FUNCTION_BLOCK NodePack_PlcBasic IMPLEMENTS I_NodePack
VAR
	nodePack_PlcBasicDisplay : NodePack_PlcBasicDisplay;
	nodePack_PlcBasicLiterals : NodePack_PlcBasicLiterals;
END_VAR

METHOD PUBLIC RegisterWithNodeFactory
VAR_INPUT
	NodeFactory : I_NodeFactory;
END_VAR
nodePack_PlcBasicDisplay.RegisterWithNodeFactory(NodeFactory);
nodePack_PlcBasicLiterals.RegisterWithNodeFactory(NodeFactory);
END_METHOD

END_FUNCTION_BLOCK

(* stored: Version 1.1.0.1, ProductVersion 3.1.4024.12
   POU NodePack_PlcBasic: Id {b1a7208c-fa6a-0ca2-104f-e5f6ddafa07d}, SpecialFunc None
   Method RegisterWithNodeFactory: Id {0a02d7c4-cf60-03c2-1373-451ec20f4e0e} *)
